Omron Sysmac Studio project distributing_station_with_timer_1.6_1 (Sysmac Studio 1.54.0.64019, StandardProject)

# Controller new_Controller_0: NJ301-1100 version 1.14
Units and slaves: Node1 : NX-ECC201 (E001); Unit 1 : NX-PC0020 (N1); Unit 2 : NX-ID5442 (N2); Unit 3 : NX-PC0010 (N3); Unit 4 : NX-PC0020 (N4); Unit 5 : NX-OD5121 (N5); Unit 6 : NX-PC0010 (N6); Power Supply : NJ-Px3001; CPU : NJ301-1100; 0 [Unit 0] : CJ1W-AD041-V1 (J01); 1 [Unit 1] : CJ1W-DA041 (J02); 2 : CJ1W-ID211 (J03); 3 : CJ1W-OC211 (J04)
Task PrimaryTask (priority 4, period or condition 1000): Program0

VAR_GLOBAL
    Station_1B2 : BOOL;  (* Ejection Cylinder Extended; at IOBus://rack#0/slot#2/Ch1_In/Ch1_In01; published *)
    Station_1B1 : BOOL;  (* Ejection Cylinder retracted; at IOBus://rack#0/slot#2/Ch1_In/Ch1_In02; published *)
    Station_2B1 : BOOL;  (* Workpiece gripped; at IOBus://rack#0/slot#2/Ch1_In/Ch1_In03; published *)
    Station_3S1 : BOOL;  (* arm_in_magazine; at IOBus://rack#0/slot#2/Ch1_In/Ch1_In04; published *)
    Station_3S2 : BOOL;  (* arm_in_downstream; at IOBus://rack#0/slot#2/Ch1_In/Ch1_In05; published *)
    Station_B4 : BOOL;  (* Magzine empty; at IOBus://rack#0/slot#2/Ch1_In/Ch1_In06; published *)
    Panel_S1 : BOOL;  (* start_button; at IOBus://rack#0/slot#2/Ch1_In/Ch1_In08; published *)
    Panel_S2 : BOOL;  (* stop_button; at IOBus://rack#0/slot#2/Ch1_In/Ch1_In09; published *)
    Panel_S4 : BOOL;  (* reset_button; at IOBus://rack#0/slot#2/Ch1_In/Ch1_In11; published *)
    Station_1Y1 : BOOL;  (* Magzine eject; at IOBus://rack#0/slot#3/Ch1_Out/Ch1_Out00; published *)
    Station_2Y1 : BOOL;  (* Vacuum on; at IOBus://rack#0/slot#3/Ch1_Out/Ch1_Out01; published *)
    Station_2Y2 : BOOL;  (* Ejector_Pulse_On; at IOBus://rack#0/slot#3/Ch1_Out/Ch1_Out02; published *)
    Station_3Y1 : BOOL;  (* arm_2_magazine; at IOBus://rack#0/slot#3/Ch1_Out/Ch1_Out03; published *)
    Station_3Y2 : BOOL;  (* arm_2_downstream; at IOBus://rack#0/slot#3/Ch1_Out/Ch1_Out04; published *)
    Station_H1 : BOOL;  (* start light; at IOBus://rack#0/slot#3/Ch1_Out/Ch1_Out08; published *)
    Station_H2 : BOOL;  (* reset light; at IOBus://rack#0/slot#3/Ch1_Out/Ch1_Out09; published *)
    Panel_H3 : BOOL;  (* Q1 light; at IOBus://rack#0/slot#3/Ch1_Out/Ch1_Out10; published *)
    Panel_H4 : BOOL;  (* Q2 light; at IOBus://rack#0/slot#3/Ch1_Out/Ch1_Out11; published *)
    Station_1B1_in : BOOL;
END_VAR

PROGRAM Program0
VAR
    FB_Panel_1 : FB_Panel;
    Panel : BOOL;
    run_mode : BOOL;
    stop_mode : BOOL;
    reset_mode : BOOL;
    FB_Actuator_T1_1 : FB_Actuator_T1;
    def : TIME;
    timer_t1 : TON;
    stat : BOOL;
    error_arm : BOOL;
    error_mode : BOOL;
    FB_Actuator_T2_1 : FB_Actuator_T2;
    error_ejec : BOOL;
    Piston : RS;
    retract_piston_int : BOOL;
END_VAR
VAR_EXTERNAL
    Station_3S1 : BOOL;
    Panel_S2 : BOOL;
    Station_3Y2 : BOOL;
    Station_3S2 : BOOL;
    Panel_S1 : BOOL;
    Station_3Y1 : BOOL;
    Panel_S4 : BOOL;
    Station_H1 : BOOL;
    Station_H2 : BOOL;
    Panel_H4 : BOOL;
    Panel_H3 : BOOL;
    Station_1B2 : BOOL;
    Station_1B1 : BOOL;
    Station_1Y1 : BOOL;
END_VAR

(* Section Section0: ladder, written here as Structured Text *)

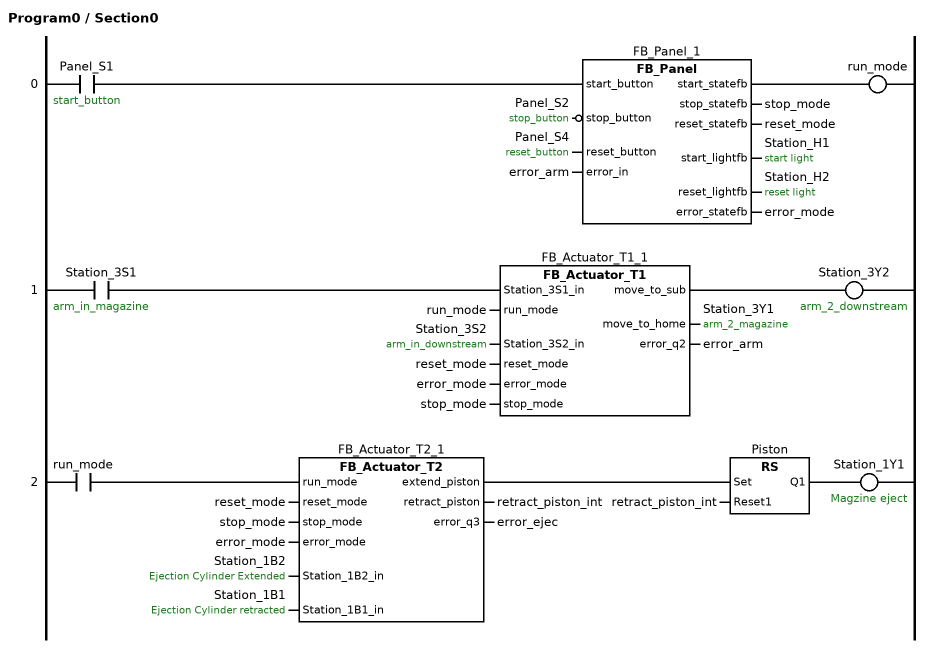
(* Rung 0 *)
FB_Panel_1(start_button := Panel_S1, stop_button := NOT Panel_S2, reset_button := Panel_S4, error_in := error_arm, stop_statefb => stop_mode, reset_statefb => reset_mode, start_lightfb => Station_H1, reset_lightfb => Station_H2, error_statefb => error_mode);
run_mode := FB_Panel_1.start_statefb;
(* Rung 1 *)
FB_Actuator_T1_1(Station_3S1_in := Station_3S1, run_mode := run_mode, Station_3S2_in := Station_3S2, reset_mode := reset_mode, error_mode := error_mode, stop_mode := stop_mode, move_to_home => Station_3Y1, error_q2 => error_arm);
Station_3Y2 := FB_Actuator_T1_1.move_to_sub;
(* Rung 2 *)
FB_Actuator_T2_1(run_mode := run_mode, reset_mode := reset_mode, stop_mode := stop_mode, error_mode := error_mode, Station_1B2_in := Station_1B2, Station_1B1_in := Station_1B1, retract_piston => retract_piston_int, error_q3 => error_ejec);
Piston(Set := FB_Actuator_T2_1.extend_piston, Reset1 := retract_piston_int);
Station_1Y1 := Piston.Q1;
END_PROGRAM

FUNCTION_BLOCK FB_Panel
VAR
    flip_flop : RS;
    flip_flop2 : RS;
    flip_flop_3 : RS;
    flip_flop3 : RS;
    stop_or_error : BOOL;
END_VAR
VAR_OUTPUT
    start_statefb : BOOL;
    stop_statefb : BOOL;
    reset_statefb : BOOL;
END_VAR
VAR_INPUT
    start_button : BOOL := False;
    stop_button : BOOL := False;
    reset_button : BOOL := False;
END_VAR
VAR_OUTPUT
    start_lightfb : BOOL;
    reset_lightfb : BOOL;
    error_statefb : BOOL;
END_VAR
VAR_INPUT
    error_in : BOOL;
END_VAR
VAR_EXTERNAL
    Panel_H4 : BOOL;
END_VAR
(* ladder, written here as Structured Text *)

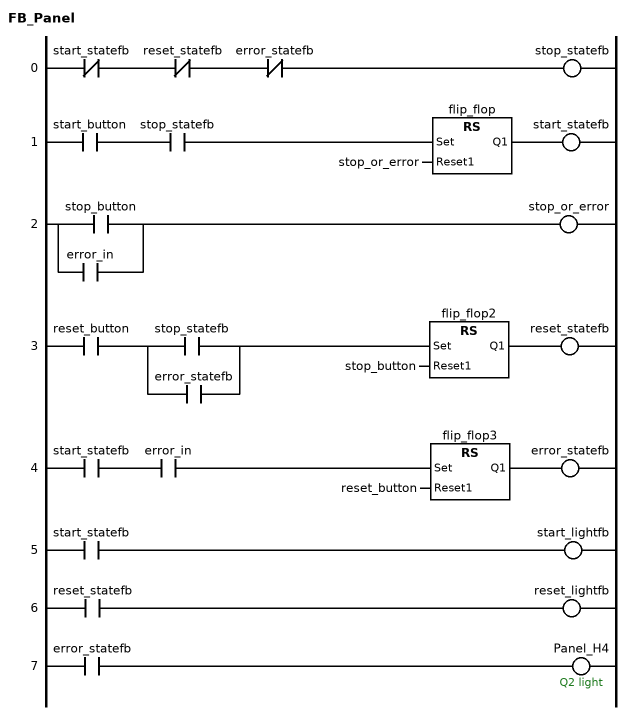
(* Rung 0 *)
stop_statefb := NOT start_statefb AND NOT reset_statefb AND NOT error_statefb;
(* Rung 1 *)
flip_flop(Set := start_button AND stop_statefb, Reset1 := stop_or_error);
start_statefb := flip_flop.Q1;
(* Rung 2 *)
stop_or_error := stop_button OR error_in;
(* Rung 3 *)
flip_flop2(Set := reset_button AND (stop_statefb OR error_statefb), Reset1 := stop_button);
reset_statefb := flip_flop2.Q1;
(* Rung 4 *)
flip_flop3(Set := start_statefb AND error_in, Reset1 := reset_button);
error_statefb := flip_flop3.Q1;
(* Rung 5 *)
start_lightfb := start_statefb;
(* Rung 6 *)
reset_lightfb := reset_statefb;
(* Rung 7 *)
Panel_H4 := error_statefb;
END_FUNCTION_BLOCK

FUNCTION_BLOCK FB_Actuator_T1
VAR
    flip_flop_1 : RS;
    flip_flop_2 : RS;
    st : BOOL;
    Panel : BOOL;
    move_to_sub_m : BOOL;
    reset_to_home : BOOL;
    timer_t1 : TON;
    flip_flop_3 : RS;
    timer_t2 : TON;
    flip_flop_4 : RS;
    error_mode_2 : BOOL;
    error_mode_1 : BOOL;
END_VAR
VAR_INPUT
    Station_3S1_in : BOOL;
    run_mode : BOOL;
    Station_3S2_in : BOOL;
    reset_mode : BOOL;
END_VAR
VAR_OUTPUT
    move_to_sub : BOOL;
    move_to_home : BOOL;
    error_q2 : BOOL;
END_VAR
VAR_INPUT
    error_mode : BOOL;
    stop_mode : BOOL;
END_VAR
VAR_EXTERNAL
    Station_3S1 : BOOL;
    Station_3Y1 : BOOL;
    Station_3S2 : BOOL;
    Station_3Y2 : BOOL;
END_VAR
(* ladder, written here as Structured Text *)

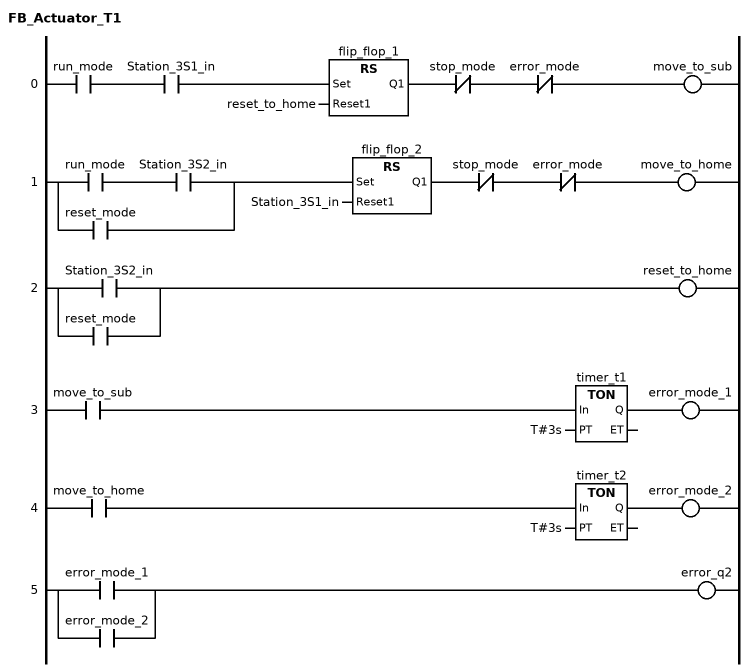
(* Rung 0 *)
flip_flop_1(Set := run_mode AND Station_3S1_in, Reset1 := reset_to_home);
move_to_sub := flip_flop_1.Q1 AND NOT stop_mode AND NOT error_mode;
(* Rung 1 *)
flip_flop_2(Set := (run_mode AND Station_3S2_in) OR reset_mode, Reset1 := Station_3S1_in);
move_to_home := flip_flop_2.Q1 AND NOT stop_mode AND NOT error_mode;
(* Rung 2 *)
reset_to_home := Station_3S2_in OR reset_mode;
(* Rung 3 *)
timer_t1(In := move_to_sub, PT := T#3s);
error_mode_1 := timer_t1.Q;
(* Rung 4 *)
timer_t2(In := move_to_home, PT := T#3s);
error_mode_2 := timer_t2.Q;
(* Rung 5 *)
error_q2 := error_mode_1 OR error_mode_2;
END_FUNCTION_BLOCK

FUNCTION_BLOCK FB_Actuator_T2
VAR
    reset_to_home : BOOL;
    retract_ff : RS;
    extend_ff : RS;
    extend_t : TON;
    retract_t : TON;
    retract_err : BOOL;
    extend_err : BOOL;
    error_eject : BOOL;
END_VAR
VAR_INPUT
    run_mode : BOOL;
    reset_mode : BOOL;
    stop_mode : BOOL;
    error_mode : BOOL;
    Station_1B2_in : BOOL;
    Station_1B1_in : BOOL;
END_VAR
VAR_OUTPUT
    extend_piston : BOOL;
    retract_piston : BOOL;
    error_q3 : BOOL;
END_VAR
(* ladder, written here as Structured Text *)

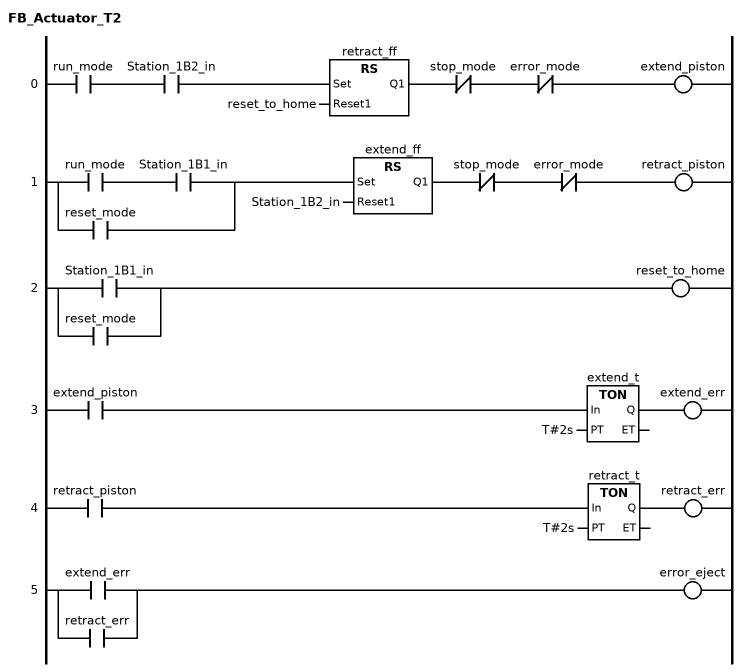
(* Rung 0 *)
retract_ff(Set := run_mode AND Station_1B2_in, Reset1 := reset_to_home);
extend_piston := retract_ff.Q1 AND NOT stop_mode AND NOT error_mode;
(* Rung 1 *)
extend_ff(Set := (run_mode AND Station_1B1_in) OR reset_mode, Reset1 := Station_1B2_in);
retract_piston := extend_ff.Q1 AND NOT stop_mode AND NOT error_mode;
(* Rung 2 *)
reset_to_home := Station_1B1_in OR reset_mode;
(* Rung 3 *)
extend_t(In := extend_piston, PT := T#2s);
extend_err := extend_t.Q;
(* Rung 4 *)
retract_t(In := retract_piston, PT := T#2s);
retract_err := retract_t.Q;
(* Rung 5 *)
error_eject := extend_err OR retract_err;
END_FUNCTION_BLOCK